FUNCTION_BLOCK PAEActValve2_Analog EXTENDS PAEActuator2way_Analog
VAR_INPUT
END_VAR
VAR_OUTPUT
END_VAR
VAR
END_VAR

METHOD PUBLIC PAEActValve2_Analog
VAR_INPUT
END_VAR
END_METHOD

END_FUNCTION_BLOCK

(* stored: Version 1.1.0.1, ProductVersion 3.1.4020.12
   POU PAEActValve2_Analog: Id {0c513952-fd68-4c45-baaf-592a4fbeeaee}, SpecialFunc None
   Method PAEActValve2_Analog: Id {1d50c705-f361-47ec-ad35-720d0c41fb0f} *)
